FUNCTION_BLOCK FB_Deadband
VAR_INPUT
	fClosedloopSignal	: LREAL;
	fVelref				: LREAL;
	fNeutral			: LREAL;
	fupperdeadband		: LREAL;
	flowerdeadband		: LREAL;
	
END_VAR
VAR_OUTPUT
	fDeadbandComp		: LREAL;
END_VAR
VAR
END_VAR

IF fVelref > 0.0 THEN
	fDeadbandComp := LIMIT(fupperdeadband,fupperdeadband + fClosedloopSignal,1.0);
ELSIF fVelref < 0.0 THEN
	fDeadbandComp := LIMIT(-1.0,flowerdeadband + fClosedloopSignal,flowerdeadband); //Kanskje minus her men tror input blir - så da blir det fikset
ELSE
	fDeadbandComp := LIMIT(-1.0,fNeutral,1.0);
END_IF

END_FUNCTION_BLOCK

(* stored: Version 1.1.0.1
   POU FB_Deadband: Id {200173d6-1190-4325-be30-42b558fdf45d}, SpecialFunc None *)
